// TIA Portal V19 export
FUNCTION_BLOCK "LEDs"   // FB15, SCL
TITLE = LED
{ S7_Optimized_Access := 'TRUE' }
AUTHOR : Siemens
// LEDs BeltLift
// stored: IsIECCheckEnabled true, MemoryReserve 100, SetENOAutomatically true
   VAR_INPUT
      startRightUp { ExternalAccessible := 'False'; ExternalVisible := 'False'; ExternalWritable := 'False'} : Bool;
      startLeftDown { ExternalAccessible := 'False'; ExternalVisible := 'False'; ExternalWritable := 'False'} : Bool;
      simulation { ExternalAccessible := 'False'; ExternalVisible := 'False'; ExternalWritable := 'False'} : Bool;
      position { ExternalAccessible := 'False'; ExternalVisible := 'False'; ExternalWritable := 'False'} : Int;
      delay { ExternalAccessible := 'False'; ExternalVisible := 'False'; ExternalWritable := 'False'} : Time := T#400ms;
   END_VAR
   VAR_OUTPUT
      leds { ExternalAccessible := 'False'; ExternalVisible := 'False'; ExternalWritable := 'False'} : Word;
   END_VAR
   VAR
      instMovingLightLift { ExternalAccessible := 'False'; ExternalVisible := 'False'; ExternalWritable := 'False'; S7_SetPoint := 'True'} : "MovingLight";
      statDirLift { ExternalAccessible := 'False'; ExternalVisible := 'False'; ExternalWritable := 'False'} : Int;
   END_VAR
   VAR CONSTANT
      STOP : Int;
      LEFT_DOWN : Int := 10;
      RIGHT_UP : Int := 20;
   END_VAR
BEGIN
   IF #simulation
   THEN
     // set led direction
     IF #startRightUp
     THEN
       #statDirLift := #RIGHT_UP;
     ELSIF #startLeftDown
     THEN
       #statDirLift := #LEFT_DOWN;
     ELSE
       #statDirLift := #STOP;
     END_IF;

     // call "MovingLight"
     #instMovingLightLift(lightDirection := #statDirLift,
                          nBitsLight := 10,
                          delay := #delay,
                          wrd1 => #leds);

   ELSE

     CASE #position OF
       0:  
         #leds := 0;
       1..10:
         #leds := 1;
       11..20:
         #leds := 2;
       21..30:
         #leds := 4;
       31..40:
         #leds := 8;
       41..50:
         #leds := 16;
       51..60:
         #leds := 32;
       61..70:
         #leds := 64;
       71..80:
         #leds := 128;
       81..90:
         #leds := 256;
       91..100:
         #leds := 512;

       ELSE  // Statement section ELSE
         #leds := 0;
     END_CASE;

   END_IF;
END_FUNCTION_BLOCK
